(* PLC project bad_wiring, plcc plcc tests 1 *)
(* stored: creationDateTime 2026-09-27T00:00:00 *)

PROGRAM Bad
  VAR
    A : BOOL;
    Q : BOOL;
  END_VAR

(* LD diagram, written out as Structured Text *)
Q := A;
(* drawn but not wired to any output: A AND *)
END_PROGRAM
